FUNCTION_BLOCK B_SECCOM_CONTROLREMOTO2 (* Basic Function Block Type *)
  (* Standard: 61499-2 *)
  (* Version 0.0, 2015-12-09, 4DIAC-IDE, 4DIAC-Consortium *)
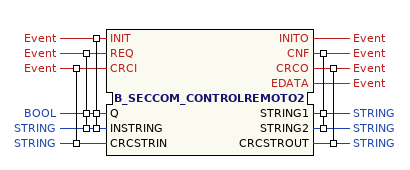
  EVENT_INPUT
    INIT WITH Q, INSTRING; (* Initialization Request *)
    REQ WITH Q, INSTRING; (* Normal Execution Request *)
    CRCI WITH CRCSTRIN;
  END_EVENT
  EVENT_OUTPUT
    INITO; (* Initialization Confirm *)
    CNF WITH STRING1, STRING2; (* Execution Confirmation *)
    CRCO WITH CRCSTROUT;
    EDATA;
  END_EVENT
  VAR_INPUT
    Q : BOOL; (* Input event qualifier *)
    INSTRING : STRING;
    CRCSTRIN : STRING;
  END_VAR
  VAR_OUTPUT
    STRING1 : STRING;
    STRING2 : STRING;
    CRCSTROUT : STRING;
  END_VAR
  VAR
    STRSUB1 : STRING; (* Internal Variable *)
    STRSUB2 : STRING; (* Internal Variable *)
    STRSUB3 : STRING; (* Internal Variable *)
    INITCONTROL : BOOL := FALSE; (* Internal Variable *)
    UINTCPY : UINT := 0; (* Internal Variable *)
  END_VAR
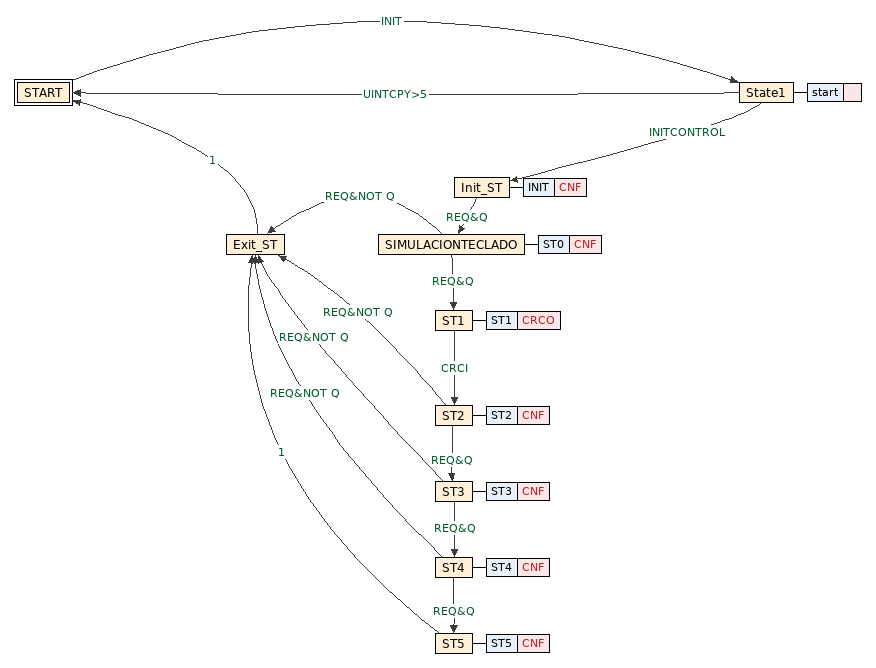
  EC_STATES
    START;
    State1 : start; (* Initial State *)
    SIMULACIONTECLADO : ST0 -> CNF;
    ST1 : ST1 -> CRCO;
    ST2 : ST2 -> CNF;
    Exit_ST;
    ST3 : ST3 -> CNF;
    ST4 : ST4 -> CNF;
    ST5 : ST5 -> CNF;
    Init_ST : INIT -> CNF;
  END_STATES
  EC_TRANSITIONS
    SIMULACIONTECLADO TO ST1 := REQ&Q;
    ST1 TO ST2 := CRCI;
    SIMULACIONTECLADO TO Exit_ST := REQ&NOT Q;
    ST2 TO ST3 := REQ&Q;
    ST2 TO Exit_ST := REQ&NOT Q;
    ST3 TO ST4 := REQ&Q;
    ST4 TO ST5 := REQ&Q;
    ST3 TO Exit_ST := REQ&NOT Q;
    ST4 TO Exit_ST := REQ&NOT Q;
    ST5 TO Exit_ST := 1;
    State1 TO Init_ST := INITCONTROL;
    Init_ST TO SIMULACIONTECLADO := REQ&Q;
    START TO State1 := INIT;
    Exit_ST TO START := 1;
    State1 TO START := UINTCPY>5;
  END_TRANSITIONS
  ALGORITHM INIT IN ST: (* Initialization algorithm *)
STRING1:='\x04\x7f';
STRING2:='\x01\x02\x03\x04';
INITCONTROL:=FALSE;
  END_ALGORITHM
  ALGORITHM ST0 IN ST: (* new algorithm *)
STRING1:='\x05';
STRING2:='\x10\x30';
  END_ALGORITHM
  ALGORITHM ST1 IN ST: (* new algorithm *)
STRSUB1:='\x01\x52\x43\x4b\x02';
STRSUB2:='\x30\x32\x09\xd6\x33\xd9';
STRSUB3:=CONCAT(STRSUB1,STRSUB2);

STRSUB2:=INSTRING;
STRSUB1:=CONCAT(STRSUB3,STRSUB2);

STRSUB2:='\xd0\x09\x03';
STRSUB3:=CONCAT(STRSUB1,STRSUB2);




CRCSTROUT:=STRSUB3;
  END_ALGORITHM
  ALGORITHM ST2 IN ST: (* new algorithm *)
STRING1:=CRCSTRIN;
STRING2:='\x10\x31';
  END_ALGORITHM
  ALGORITHM ST3 IN ST: (* new algorithm *)
STRING1:='\x04';
STRING2:='\x05\x7f';
  END_ALGORITHM
  ALGORITHM ST4 IN ST: (* new algorithm *)
STRING1:='\x10\x30';
STRING2:='\x02\x03';
  END_ALGORITHM
  ALGORITHM ST5 IN ST: (* new algorithm *)
STRING1:='\x10\x31';
STRING2:='\x04\x7f';
  END_ALGORITHM
  ALGORITHM start IN ST: (* new algorithm *)
INITCONTROL:=TRUE;
  END_ALGORITHM
  ALGORITHM PE1 IN ST: (* new algorithm *)
STRSUB1:='\x01\x52\x43\x4b\x02';
STRSUB2:='\x30\x31';
STRSUB3:=CONCAT(STRSUB1,STRSUB2);

STRSUB2:='\x03';
STRSUB1:=CONCAT(STRSUB3,STRSUB2);

CRCSTROUT:=STRSUB1;
  END_ALGORITHM
  ALGORITHM PE2 IN ST: (* new algorithm *)
STRING1:=CRCSTRIN;
STRING2:='\x10\x31';
  END_ALGORITHM
  ALGORITHM PE3 IN ST: (* new algorithm *)
STRING1:='\x04';
STRING2:='\x05\x7f';
  END_ALGORITHM
  ALGORITHM PE4 IN ST: (* new algorithm *)
STRING1:='\x10\x30';
STRING2:='\x02\x03';
  END_ALGORITHM
  ALGORITHM PE5 IN ST: (* new algorithm *)
STRING1:='\x10\x31';
STRING2:='\x04\x7f';
  END_ALGORITHM
  ALGORITHM IT1 IN ST: (* new algorithm *)
STRSUB1:='\x01\x52\x43\x4b\x02';
STRSUB2:='\x31\x31';
STRSUB3:=CONCAT(STRSUB1,STRSUB2);

STRSUB2:='\x03';
STRSUB1:=CONCAT(STRSUB3,STRSUB2);

CRCSTROUT:=STRSUB1;
  END_ALGORITHM
  ALGORITHM LE1 IN ST: (* new algorithm *)
STRSUB1:='\x01\x52\x43\x4b\x02';
STRSUB2:='\x31\x30';
STRSUB3:=CONCAT(STRSUB1,STRSUB2);

STRSUB2:='\x03';
STRSUB1:=CONCAT(STRSUB3,STRSUB2);

CRCSTROUT:=STRSUB1;
  END_ALGORITHM
  ALGORITHM IE40 IN ST: (* new algorithm *)
DATA:=RDATA;
  END_ALGORITHM
  ALGORITHM IT50 IN ST: (* new algorithm *)
DATA:=RDATA;
  END_ALGORITHM
  ALGORITHM LE50 IN ST: (* new algorithm *)
DATA:=RDATA;
  END_ALGORITHM
  ALGORITHM PE50 IN ST: (* new algorithm *)
DATA:=RDATA;
  END_ALGORITHM
END_FUNCTION_BLOCK
